FUNCTION_BLOCK FB_CNMachineSystem
VAR_INPUT
END_VAR
VAR_OUTPUT
END_VAR
VAR
END_VAR

END_FUNCTION_BLOCK

(* stored: Version 1.1.0.1, ProductVersion 3.1.4024.10
   POU FB_CNMachineSystem: Id {f6a8ead8-0d82-4b08-9375-be8afa66c1f4}, SpecialFunc None *)
